KUKA KRL program: saco_5_m4.src, saco_5_m4.dat

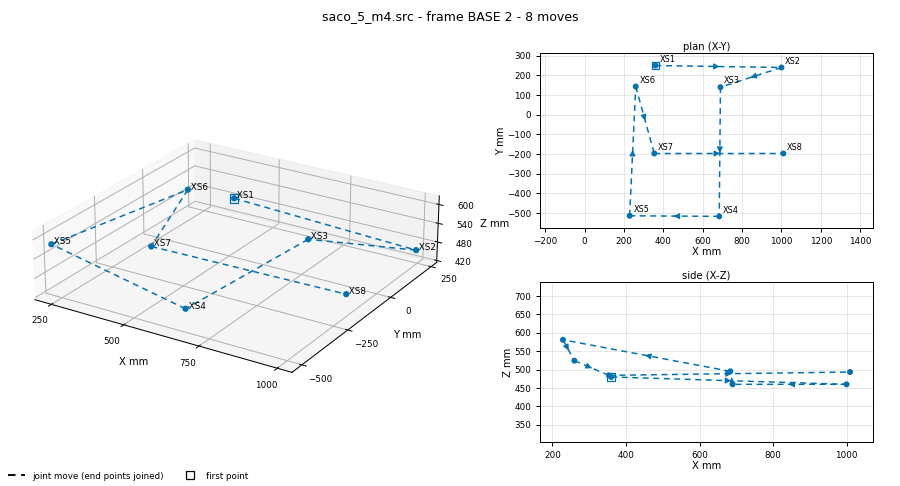
[picture p0: tool path of saco_5_m4.src in frame BASE 2, 8 of 16 moves have a stored position in this frame; points joined in program order, loops and branches not executed]
--- saco_5_m4.src ---
&ACCESS RVP1
&REL 9
&PARAM DISKPATH = KRC:\R1\Program\SACO_5
&PARAM TEMPLATE = C:\KRC\Roboter\Template\vorgabe
&PARAM EDITMASK = *
DEF saco_5_m4( )
;Fold DECLARACION VARIABLES
DECL E6POS POS_A
DECL E6POS POS_B
DECL E6POS POS_C
DECL REAL INC_Z
DECL INT PLANTA
DECL INT SACOS_A_PALETIZAR
DECL E6POS PUNTO[20]
DECL INT n
EXT COGE_5 ()
;Endfold
;FOLD INI;%{PE}
  ;FOLD BASISTECH INI
    GLOBAL INTERRUPT DECL 3 WHEN $STOPMESS==TRUE DO IR_STOPM ( )
    INTERRUPT ON 3
    BAS (#INITMOV,0 )
  ;ENDFOLD (BASISTECH INI)
;FOLD SPOTTECH INI
USERSPOT(#INIT)
;ENDFOLD (SPOTTECH INI)
;FOLD GRIPPERTECH INI
USER_GRP(0,DUMMY,DUMMY,GDEFAULT)
;ENDFOLD (GRIPPERTECH INI)
  ;FOLD USER INI
    ;Make your modifications here

  ;ENDFOLD (USER INI)
;ENDFOLD (INI)
; === PROGRAMA 200 SACOS 5 KG MOSAICO 10-10 ==
;Fold VARIABLES
INC_Z=0  ;Cota Inicial
PLANTA = 0
N_SACO=0
SACOS_A_PALETIZAR=200
n=1
PUNTO[1]=XP1
PUNTO[2]=XP2
PUNTO[3]=XP3
PUNTO[4]=XP4
PUNTO[5]=XP5
PUNTO[6]=XP6
PUNTO[7]=XP7
PUNTO[8]=XP8
PUNTO[9]=XP9
PUNTO[10]=XP10
PUNTO[11]=XP11
PUNTO[12]=XP12
PUNTO[13]=XP13
PUNTO[14]=XP14
PUNTO[15]=XP15
PUNTO[16]=XP16
PUNTO[17]=XP17
PUNTO[18]=XP18
PUNTO[19]=XP19
PUNTO[20]=XP20
;Endfold
;FOLD PTP HOME  Vel= 100 % DEFAULT;%{PE}%MKUKATPBASIS,%CMOVE,%VPTP,%P 1:PTP, 2:HOME, 3:, 5:100, 7:DEFAULT
$BWDSTART = FALSE
PDAT_ACT=PDEFAULT
FDAT_ACT=FHOME
BAS (#PTP_PARAMS,100 )
$H_POS=XHOME
PTP  XHOME
;ENDFOLD
;Fold Compruebo Palet
WAIT FOR PALET_LIBRE OR SALIR_PROGRAMA_ACTUAL
IF SALIR_PROGRAMA_ACTUAL == TRUE THEN
   PULSE ( OK_LEIDO_SALIR_PROGRAMA, true, 0.5 )
   WAIT SEC 1
   GOTO SALIRPROG
ENDIF
;Endfold

BOMBA =TRUE
;=== BUCLE PRINCIPAL ==
FOR PLANTA=0 TO 30 ;Bucle de plantas

FOR n=1 TO 20 ;Bucle de sacos
SACO:

;Fold WAIT FOR REPITE_SACO: Espero repetir saco si ha caido
IF (ERROR_SACO_CAIDO == TRUE ) THEN
   WAIT FOR REPITE_SACO OR SALIR_PROGRAMA_ACTUAL
   ERROR_SACO_CAIDO = FALSE
ENDIF
;Endfold
COGE_5 () ;Llamo programa coger
;Fold CONDICION DE SALIDA DE PROGRAMA PLC
IF SALIR == TRUE THEN
   GOTO SALIRPROG
ENDIF
;Endfold

;Fold DEFINICION PUNTOS AUXILIARES
POS_A =PUNTO[n]
POS_B =PUNTO[n]
POS_C =PUNTO[n]

POS_A.Z=POS_A.Z+INC_Z+400
POS_B.Z=POS_B.Z+INC_Z+250
POS_C.Z=POS_C.Z+INC_Z+60

;Endfold

BAS(#BASE,2) ;Cambio de base
$APO.CPTP = 70


;Fold Velocidad SACO5
FOR ax_num=1 TO 6
$VEL_AXIS[ax_num]=vptpSACO5
$ACC_AXIS[ax_num]=vaccSACO5
ENDFOR
$VEL.CP=vlinSACO5
;Endfold
PTP POS_A C_PTP
;Fold Velocidad Media
FOR ax_num=1 TO 6
$VEL_AXIS[ax_num]=vptpM
$ACC_AXIS[ax_num]=vaccM
ENDFOR
$VEL.CP=vlinM
;Endfold
PTP POS_B C_PTP
;Fold Velocidad Lenta
FOR ax_num=1 TO 6
$VEL_AXIS[ax_num]=vptpL
$ACC_AXIS[ax_num]=vaccL
ENDFOR
$VEL.CP=vlinL
;Endfold
LIN POS_C
;Fold Compruebo caida de saco
IF (VACOESTATO == FALSE) THEN ;Condicion de saco perdido
   ERROR_SACO_CAIDO = TRUE
   FOR ax_num=1 TO 6
   $VEL_AXIS[ax_num]=vptpR
   $ACC_AXIS[ax_num]=vaccR
   ENDFOR
   $VEL.CP=vlinR
   LIN POS_A
   ;FOLD PTP HOME  Vel= 100 % DEFAULT;%{PE}%MKUKATPBASIS,%CMOVE,%VPTP,%P 1:PTP, 2:HOME, 3:, 5:100, 7:DEFAULT
$BWDSTART = FALSE
PDAT_ACT=PDEFAULT
FDAT_ACT=FHOME
BAS (#PTP_PARAMS,100 )
$H_POS=XHOME
PTP  XHOME
;ENDFOLD
   GOTO SACO
ENDIF
;Endfold

WAIT SEC 0.2
VACIO=FALSE  ;Abro vacio
WAIT FOR NOT VACOESTATO OR VOLVER_COGER ;Espero Vacoestato

;Fold Velocidad Rapida
Continue
FOR ax_num=1 TO 6
$VEL_AXIS[ax_num]=vptpR
$ACC_AXIS[ax_num]=vaccR
ENDFOR
$VEL.CP=vlinR
;Endfold

LIN POS_A C_DIS

;Fold Incremento Saco
N_SACO=N_SACO+1
IF (N_SACO >= SACOS_A_PALETIZAR) THEN
   GOTO FINAL
ENDIF
;Endfold

ENDFOR

;Fold Incremento Planta
PLANTA = PLANTA + 1

INC_Z=INC_Z+95.0  ;Incremento cota superior

;Endfold

ENDFOR

GOTO FINAL
;Fold PUNTOS COGIDA SOLO PARA MODIFICAR TOUCHAP

;FOLD PTP S1 Vel=50 % PDAT1 Tool[1]:VENTOSA_SACOS Base[2]:PALETS;%{PE}%R 8.2.24,%MKUKATPBASIS,%CMOVE,%VPTP,%P 1:PTP, 2:S1, 3:, 5:50, 7:PDAT1
$BWDSTART=FALSE
PDAT_ACT=PPDAT1
FDAT_ACT=FS1
BAS(#PTP_PARAMS,50)
PTP XS1
;ENDFOLD
;FOLD PTP S2 Vel=50 % PDAT2 Tool[1]:VENTOSA_SACOS Base[2]:PALETS;%{PE}%R 8.2.24,%MKUKATPBASIS,%CMOVE,%VPTP,%P 1:PTP, 2:S2, 3:, 5:50, 7:PDAT2
$BWDSTART=FALSE
PDAT_ACT=PPDAT2
FDAT_ACT=FS2
BAS(#PTP_PARAMS,50)
PTP XS2
;ENDFOLD
;FOLD PTP S3 Vel=50 % PDAT3 Tool[1]:VENTOSA_SACOS Base[2]:PALETS;%{PE}%R 8.2.24,%MKUKATPBASIS,%CMOVE,%VPTP,%P 1:PTP, 2:S3, 3:, 5:50, 7:PDAT3
$BWDSTART=FALSE
PDAT_ACT=PPDAT3
FDAT_ACT=FS3
BAS(#PTP_PARAMS,50)
PTP XS3
;ENDFOLD
;FOLD PTP S4 Vel=50 % PDAT4 Tool[1]:VENTOSA_SACOS Base[2]:PALETS;%{PE}%R 8.2.24,%MKUKATPBASIS,%CMOVE,%VPTP,%P 1:PTP, 2:S4, 3:, 5:50, 7:PDAT4
$BWDSTART=FALSE
PDAT_ACT=PPDAT4
FDAT_ACT=FS4
BAS(#PTP_PARAMS,50)
PTP XS4
;ENDFOLD
;planta2
;FOLD PTP S5 Vel=50 % PDAT5 Tool[1]:VENTOSA_SACOS Base[2]:PALETS;%{PE}%R 8.2.24,%MKUKATPBASIS,%CMOVE,%VPTP,%P 1:PTP, 2:S5, 3:, 5:50, 7:PDAT5
$BWDSTART=FALSE
PDAT_ACT=PPDAT5
FDAT_ACT=FS5
BAS(#PTP_PARAMS,50)
PTP XS5
;ENDFOLD
;FOLD PTP S6 Vel=50 % PDAT6 Tool[1]:VENTOSA_SACOS Base[2]:PALETS;%{PE}%R 8.2.24,%MKUKATPBASIS,%CMOVE,%VPTP,%P 1:PTP, 2:S6, 3:, 5:50, 7:PDAT6
$BWDSTART=FALSE
PDAT_ACT=PPDAT6
FDAT_ACT=FS6
BAS(#PTP_PARAMS,50)
PTP XS6
;ENDFOLD
;FOLD PTP S7 Vel=50 % PDAT7 Tool[1]:VENTOSA_SACOS Base[2]:PALETS;%{PE}%R 8.2.24,%MKUKATPBASIS,%CMOVE,%VPTP,%P 1:PTP, 2:S7, 3:, 5:50, 7:PDAT7
$BWDSTART=FALSE
PDAT_ACT=PPDAT7
FDAT_ACT=FS7
BAS(#PTP_PARAMS,50)
PTP XS7
;ENDFOLD
;FOLD PTP S8 Vel=50 % PDAT8 Tool[1]:VENTOSA_SACOS Base[2]:PALETS;%{PE}%R 8.2.24,%MKUKATPBASIS,%CMOVE,%VPTP,%P 1:PTP, 2:S8, 3:, 5:50, 7:PDAT8
$BWDSTART=FALSE
PDAT_ACT=PPDAT8
FDAT_ACT=FS8
BAS(#PTP_PARAMS,50)
PTP XS8
;ENDFOLD
;Endfold
FINAL:

PULSE ( PALET_COMPLETO, TRUE, 0.5 )
WAIT SEC 1

SALIRPROG:

N_SACO=0
SALIR=FALSE
BOMBA=FALSE

;FOLD PTP HOME CONT Vel=ptpM % DEFAULT;%{PE}%R 8.2.24,%MKUKATPBASIS,%CMOVE,%VPTP,%P 1:PTP, 2:HOME, 3:C_DIS, 5:50, 7:DEFAULT
$BWDSTART=FALSE
PDAT_ACT=PDEFAULT
FDAT_ACT=FHOME
BAS(#PTP_PARAMS,vptpM)
$H_POS=XHOME
$APO.CPTP = 70
PTP XHOME C_PTP
;ENDFOLD

END

--- saco_5_m4.dat ---
&ACCESS RVP1
&REL 9
&PARAM DISKPATH = KRC:\R1\Program\SACO_5
&PARAM TEMPLATE = C:\KRC\Roboter\Template\vorgabe
&PARAM EDITMASK = *
DEFDAT  saco_5_m4
;FOLD EXTERNAL DECLARATIONS;%{PE}%MKUKATPBASIS,%CEXT,%VCOMMON,%P
;FOLD GRIPPERTECH EXT
EXT  H50 (INT  :IN,INT  :IN,INT  :IN,GRP_TYP  :IN )
;ENDFOLD (GRIPPERTECH EXT)
;FOLD SPOTTECH EXT
EXT  USERSPOT (S_COMMAND  :IN,SPOT_TYPE  :IN )
;ENDFOLD (SPOTTECH EXT)
;FOLD BASISTECH EXT;%{PE}%MKUKATPBASIS,%CEXT,%VEXT,%P
EXT  BAS (BAS_COMMAND  :IN,REAL  :IN )
DECL INT SUCCESS
;ENDFOLD (BASISTECH EXT)
;FOLD USER EXT;%{E}%MKUKATPUSER,%CEXT,%VEXT,%P
;Make your modifications here

;ENDFOLD (USER EXT)
;ENDFOLD (EXTERNAL DECLARATIONS)
DECL BASIS_SUGG_T LAST_BASIS={POINT1[] "S28                     ",POINT2[] "S28                     ",CP_PARAMS[] "CPDAT0                  ",PTP_PARAMS[] "PDAT28                  ",CONT[] "                        ",CP_VEL[] "2.0                     ",PTP_VEL[] "50                      ",SYNC_PARAMS[] "SYNCDAT                 ",SPL_NAME[] "S0                      "}

DECL E6POS XS1={X 359.99649,Y 249.997894,Z 480.002411,A 86.8255005,B 0.369327009,C -179.812195,S 2,T 35,E1 0.0,E2 0.0,E3 0.0,E4 0.0,E5 0.0,E6 0.0}
DECL FDAT FS1={TOOL_NO 1,BASE_NO 2,IPO_FRAME #BASE,POINT2[] " ",TQ_STATE FALSE}
DECL PDAT PPDAT1={VEL 100.0,ACC 100.0,APO_DIST 100.0,APO_MODE #CDIS,GEAR_JERK 50.0}
DECL E6POS XS2={X 999.999878,Y 240.001907,Z 459.999786,A -92.3902283,B -0.366795003,C 179.807404,S 2,T 3,E1 0.0,E2 0.0,E3 0.0,E4 0.0,E5 0.0,E6 0.0}
DECL FDAT FS2={TOOL_NO 1,BASE_NO 2,IPO_FRAME #BASE,POINT2[] " ",TQ_STATE FALSE}
DECL PDAT PPDAT2={VEL 100.0,ACC 100.0,APO_DIST 100.0,APO_MODE #CDIS,GEAR_JERK 50.0}
DECL E6POS XS3={X 689.999573,Y 140.003296,Z 459.99469,A -2.77452111,B 0.190423205,C 179.632004,S 2,T 35,E1 0.0,E2 0.0,E3 0.0,E4 0.0,E5 0.0,E6 0.0}
DECL FDAT FS3={TOOL_NO 1,BASE_NO 2,IPO_FRAME #BASE,POINT2[] " ",TQ_STATE FALSE}
DECL PDAT PPDAT3={VEL 100.0,ACC 100.0,APO_DIST 100.0,APO_MODE #CDIS,GEAR_JERK 50.0}
DECL E6POS XS4={X 683.710205,Y -516.212585,Z 495.420593,A 177.664795,B -0.192770898,C -179.633194,S 2,T 11,E1 0.0,E2 0.0,E3 0.0,E4 0.0,E5 0.0,E6 0.0}
DECL FDAT FS4={TOOL_NO 1,BASE_NO 2,IPO_FRAME #BASE,POINT2[] " ",TQ_STATE FALSE}
DECL PDAT PPDAT4={VEL 100.0,ACC 100.0,APO_DIST 100.0,APO_MODE #CDIS,GEAR_JERK 50.0}

DECL E6POS XS5={X 228.594498,Y -513.38562,Z 581.090027,A 178.337296,B -0.197238594,C -179.635498,S 2,T 11,E1 0.0,E2 0.0,E3 0.0,E4 0.0,E5 0.0,E6 0.0}
DECL FDAT FS5={TOOL_NO 1,BASE_NO 2,IPO_FRAME #BASE,POINT2[] " ",TQ_STATE FALSE}
DECL PDAT PPDAT5={VEL 100.0,ACC 100.0,APO_DIST 100.0,APO_MODE #CDIS,GEAR_JERK 50.0}
DECL E6POS XS6={X 259.555908,Y 143.434494,Z 524.370605,A -3.0096159,B 0.188729897,C 179.631104,S 2,T 35,E1 0.0,E2 0.0,E3 0.0,E4 0.0,E5 0.0,E6 0.0}
DECL FDAT FS6={TOOL_NO 1,BASE_NO 2,IPO_FRAME #BASE,POINT2[] " ",TQ_STATE FALSE}
DECL PDAT PPDAT6={VEL 100.0,ACC 100.0,APO_DIST 100.0,APO_MODE #CDIS,GEAR_JERK 50.0}
DECL E6POS XS7={X 353.689789,Y -196.9095,Z 484.410004,A 86.8238068,B 0.3691881,C -179.811996,S 2,T 43,E1 0.0,E2 0.0,E3 0.0,E4 0.0,E5 0.0,E6 0.0}
DECL FDAT FS7={TOOL_NO 1,BASE_NO 2,IPO_FRAME #BASE,POINT2[] " ",TQ_STATE FALSE}
DECL PDAT PPDAT7={VEL 100.0,ACC 100.0,APO_DIST 100.0,APO_MODE #CDIS,GEAR_JERK 50.0}
DECL E6POS XS8={X 1009.48798,Y -196.910294,Z 493.416199,A -93.0203171,B -0.3688972,C 179.811401,S 2,T 3,E1 0.0,E2 0.0,E3 0.0,E4 0.0,E5 0.0,E6 0.0}
DECL FDAT FS8={TOOL_NO 1,BASE_NO 2,IPO_FRAME #BASE,POINT2[] " ",TQ_STATE FALSE}
DECL PDAT PPDAT8={VEL 100.0,ACC 100.0,APO_DIST 100.0,APO_MODE #CDIS,GEAR_JERK 50.0}

;PUNTOS NUEVOS

;Planta 0
DECL E6POS XP1 ={X 360 ,Y  220,Z 400,A 86.8255005,B 0.369327009,C -179.812195,S 2,T 35,E1 0.0,E2 0.0,E3 0.0,E4 0.0,E5 0.0,E6 0.0}
DECL E6POS XP2 ={X 360 ,Y  -60,Z 400,A 86.8255005,B 0.369327009,C -179.812195,S 2,T 35,E1 0.0,E2 0.0,E3 0.0,E4 0.0,E5 0.0,E6 0.0}
DECL E6POS XP3 ={X 360 ,Y -340,Z 400,A 86.8255005,B 0.369327009,C -179.812195,S 2,T 35,E1 0.0,E2 0.0,E3 0.0,E4 0.0,E5 0.0,E6 0.0}
DECL E6POS XP4 ={X 360 ,Y -620,Z 400,A 86.8255005,B 0.369327009,C -179.812195,S 2,T 35,E1 0.0,E2 0.0,E3 0.0,E4 0.0,E5 0.0,E6 0.0}

DECL E6POS XP5 ={X 1000,Y  240,Z 400,A -92.3902283,B -0.366795003,C 179.807404,S 2,T 3,E1 0.0,E2 0.0,E3 0.0,E4 0.0,E5 0.0,E6 0.0}
DECL E6POS XP6 ={X 1000,Y  -40,Z 400,A -92.3902283,B -0.366795003,C 179.807404,S 2,T 3,E1 0.0,E2 0.0,E3 0.0,E4 0.0,E5 0.0,E6 0.0}
DECL E6POS XP7 ={X 1000,Y -320,Z 400,A -92.3902283,B -0.366795003,C 179.807404,S 2,T 3,E1 0.0,E2 0.0,E3 0.0,E4 0.0,E5 0.0,E6 0.0}
DECL E6POS XP8 ={X 1000,Y -600,Z 400,A -92.3902283,B -0.366795003,C 179.807404,S 2,T 3,E1 0.0,E2 0.0,E3 0.0,E4 0.0,E5 0.0,E6 0.0}

DECL E6POS XP9 ={X 690 ,Y  140,Z 400,A -2.77452111,B 0.190423205,C 179.632004,S 2,T 35,E1 0.0,E2 0.0,E3 0.0,E4 0.0,E5 0.0,E6 0.0}
DECL E6POS XP10={X 680 ,Y -520,Z 400,A 177.664795,B -0.192770898,C -179.633194,S 2,T 11,E1 0.0,E2 0.0,E3 0.0,E4 0.0,E5 0.0,E6 0.0}

;Planta 1
DECL E6POS XP11={X 260 ,Y -510,Z 500,A 178.337296,B -0.197238594,C -179.635498,S 2,T 11,E1 0.0,E2 0.0,E3 0.0,E4 0.0,E5 0.0,E6 0.0}
DECL E6POS XP12={X 540 ,Y -510,Z 500,A 178.337296,B -0.197238594,C -179.635498,S 2,T 11,E1 0.0,E2 0.0,E3 0.0,E4 0.0,E5 0.0,E6 0.0}
DECL E6POS XP13={X 820 ,Y -510,Z 500,A 178.337296,B -0.197238594,C -179.635498,S 2,T 11,E1 0.0,E2 0.0,E3 0.0,E4 0.0,E5 0.0,E6 0.0}
DECL E6POS XP14={X 1110,Y -510,Z 500,A 178.337296,B -0.197238594,C -179.635498,S 2,T 11,E1 0.0,E2 0.0,E3 0.0,E4 0.0,E5 0.0,E6 0.0}

DECL E6POS XP15={X 260 ,Y 140,Z 500,A -3.0096159,B 0.188729897,C 179.631104,S 2,T 35,E1 0.0,E2 0.0,E3 0.0,E4 0.0,E5 0.0,E6 0.0}
DECL E6POS XP16={X 540 ,Y 140,Z 500,A -3.0096159,B 0.188729897,C 179.631104,S 2,T 35,E1 0.0,E2 0.0,E3 0.0,E4 0.0,E5 0.0,E6 0.0}
DECL E6POS XP17={X 820 ,Y 140,Z 500,A -3.0096159,B 0.188729897,C 179.631104,S 2,T 35,E1 0.0,E2 0.0,E3 0.0,E4 0.0,E5 0.0,E6 0.0}
DECL E6POS XP18={X 1100,Y 140,Z 500,A -3.0096159,B 0.188729897,C 179.631104,S 2,T 35,E1 0.0,E2 0.0,E3 0.0,E4 0.0,E5 0.0,E6 0.0}

DECL E6POS XP19={X 350 ,Y -200,Z 500,A 86.8238068,B 0.3691881,C -179.811996,S 2,T 43,E1 0.0,E2 0.0,E3 0.0,E4 0.0,E5 0.0,E6 0.0}
DECL E6POS XP20={X 1000,Y -200,Z 500,A -93.0203171,B -0.3688972,C 179.811401,S 2,T 3,E1 0.0,E2 0.0,E3 0.0,E4 0.0,E5 0.0,E6 0.0}

ENDDAT
